FUNCTION_BLOCK FB_Year EXTENDS FB_Object IMPLEMENTS I_SeasonControl, I_CyclicTask
VAR
    fbSeasonStateMachine:   FB_SeasonStateMachine(THIS^);
    fbWinter:               FB_Winter(THIS^, THIS^.fbSeasonStateMachine);
    fbSpring:               FB_Spring(THIS^, THIS^.fbSeasonStateMachine);
    fbSummer:               FB_Summer(THIS^, THIS^.fbSeasonStateMachine);
    fbAutumn:               FB_Autumn(THIS^, THIS^.fbSeasonStateMachine);

    nCounter:               UDINT;
    nModVal:                UDINT := 500;
END_VAR

METHOD ChangeToSummerTyres
VAR_INPUT
END_VAR
THIS^.CurrentState().ChangeToSummerTyres();
END_METHOD

METHOD ChangeToWinterTyres
VAR_INPUT
END_VAR
THIS^.CurrentState().ChangeToWinterTyres();
END_METHOD

METHOD CurrentState : I_SeasonState
__QUERYINTERFACE(THIS^.fbSeasonStateMachine.ipState, CurrentState);
END_METHOD

METHOD FB_init : BOOL
VAR_INPUT
    bInitRetains:           BOOL; // if TRUE, the retain variables are initialized (warm start / cold start)
    bInCopyCode:            BOOL;  // if TRUE, the instance afterwards gets moved into the copy code (online change)
    ipParentObject:         I_Object;
END_VAR
THIS^.fbSeasonStateMachine.SetState(THIS^.StateSummer);
THIS^.CurrentState().ChangeToSummerTyres();
END_METHOD

METHOD NextSeason
VAR_INPUT
END_VAR
THIS^.fbSeasonStateMachine.NextSeason();
END_METHOD

METHOD Run
VAR_INPUT
END_VAR
THIS^.nCounter := THIS^.nCounter + 1;
THIS^.fbSeasonStateMachine.Run();
END_METHOD

PROPERTY StateAutumn : I_State
GET
StateAutumn := THIS^.fbAutumn;
END_GET
END_PROPERTY

PROPERTY StateSpring : I_State
GET
StateSpring := THIS^.fbSpring;
END_GET
END_PROPERTY

PROPERTY StateSummer : I_State
GET
StateSummer := THIS^.fbSummer;
END_GET
END_PROPERTY

PROPERTY StateWinter : I_State
GET
StateWinter := THIS^.fbWinter;
END_GET
END_PROPERTY

END_FUNCTION_BLOCK

(* stored: Version 1.1.0.1, ProductVersion 3.1.4024.12
   POU FB_Year: Id {ab586e98-5688-4741-8fa9-f6f036cb2866}, SpecialFunc None
   Folder Properties: Id {bb0847b0-23d8-456c-8023-595a9f24d8b6}
   Method ChangeToSummerTyres: Id {25d6f496-e955-4f0e-b98a-8b121601874b}
   Method ChangeToWinterTyres: Id {7590e57a-24dd-44e0-abcf-7d819aa5eb88}
   Method CurrentState: Id {c8e36b6e-0333-4c2b-9b53-bb47a49de1bd}
   Method FB_init: Id {c50045c6-dd1c-444f-ad22-0c9361c175f5}
   Method NextSeason: Id {99bad3ac-ffd2-4027-9407-a43b26b4d98f}
   Method Run: Id {301a778b-ea2d-427d-a14f-15f72d0fbede}
   Property StateAutumn: Id {7b203f93-e055-4c78-b941-b99a6f21a042}
   Get Get: Id {39499a01-2973-4cae-93cc-98008e1f4c8a}
   Property StateSpring: Id {627552e2-b920-493a-88d5-7d59040dc7e2}
   Get Get: Id {ba247c47-7b27-4237-9619-f829b640bbd0}
   Property StateSummer: Id {98e1a874-7502-49a9-ad52-d8f7c20f7ae8}
   Get Get: Id {199d7976-d4e2-49a9-b221-1ac9c0f88a2b}
   Property StateWinter: Id {3e4406a0-98f9-4620-b332-248e18bd0370}
   Get Get: Id {db59fa05-40b3-4ce8-93a7-dd1d5ec2931a} *)
